(* IEC 61131-3 sources: ics/BLR1_PhoenixContact/BLR1_AXC1050_21/LogicalPOUs/AIO, 3 files *)

(* ---- SensorFB.ST ---- *)
(*@PROPERTIES_EX@
TYPE: POU
LOCALE: 0
IEC_LANGUAGE: ST
PLC_TYPE: independent
PROC_TYPE: independent
GROUP: AIO.FB
*)
(*@KEY@:DESCRIPTION*)

(*@KEY@:END_DESCRIPTION*)
FUNCTION_BLOCK SensorFB

(*Group:Default*)

VAR_IN_OUT
    Snsr_strct :	SNSR;
END_VAR

VAR
    RealValue :	REAL;
    bar_kgf :	REAL;
END_VAR

VAR_IN_OUT
    Buff :	SNSR_BUFF;
END_VAR

VAR
    SumValue :	REAL;
    y :	INT;
    INIT :	BOOL;
    FltrValue :	REAL;
    x :	INT;
END_VAR

VAR_OUTPUT
    Event :	SNSR_EVENT;
END_VAR

VAR_IN_OUT
    Aux_strct :	SNSR_MISC;
END_VAR

VAR_EXTERNAL
    TICK_100MS_PLS :	BOOL;
END_VAR

(*@KEY@: WORKSHEET
NAME: SensorFB
IEC_LANGUAGE: ST
*)

(*============================================================================*)
(*Fault operation & converting PIW to real value*)
(*============================================================================*)
IF (Snsr_strct.PIW < 0) OR (Snsr_strct.PIW > Snsr_strct.ADC_Range) OR
    Snsr_strct.CW.ExtFault OR (Snsr_strct.DiagCode > word#16#8000) THEN         (*Snsr_strct Failed*)
    Snsr_strct.SW.Fault:= TRUE;
    RealValue:= 0.0;
ELSE                                                                            (*Snsr_strct OK*)
    IF Snsr_strct.ADC_Range <= 0 THEN
        Snsr_strct.ADC_Range:= 1;
    END_IF;
    Snsr_strct.SW.Fault:= FALSE;
    RealValue:= (Snsr_strct.Ymax - Snsr_strct.Ymin) * bar_kgf *
        INT_TO_REAL(Snsr_strct.PIW) / INT_TO_REAL(Snsr_strct.ADC_Range) +
        Snsr_strct.Ymin ;
END_IF;

(*============================================================================*)
(*Converting from bar to kgf/sm2*)
(*============================================================================*)
IF Snsr_strct.CW.bar_kgf THEN
    bar_kgf:= 1.0197;
ELSE
    bar_kgf:= 1.0;
END_IF;

(*============================================================================*)
(*SMA filter operation*)
(*============================================================================*)
IF INIT THEN
    IF TICK_100MS_PLS THEN
        Aux_strct.SamplingTickCount:= Aux_strct.SamplingTickCount + 1;
    END_IF;
ELSE
    Aux_strct.SamplingTickCount:= 0;
END_IF;

IF Snsr_strct.CW.FltrEn THEN
    IF NOT INIT THEN                                                            (*Initialization*)
        FOR y:= 0 TO 9 DO
            Buff[y]:= RealValue;
            SumValue:= SumValue + Buff[y];
        END_FOR;
        INIT:= TRUE;
    ELSE
        IF Aux_strct.SamplingTickCount >= (Snsr_strct.SamplingTime * 10) THEN   (*Buffer shIFting AND changing last element*)
            FOR y:= 0 TO 8 DO
                x:= y + 1;
                Buff[y]:= Buff[x];
            END_FOR;
            Buff[9]:= RealValue;
            SumValue:= SumValue + RealValue - Buff[0];
            Aux_strct.SamplingTickCount:= 0;
        END_IF;
        FltrValue:= SumValue / 10.0;
    END_IF;
ELSE
    INIT:= FALSE;
    SumValue:= 0.0;
    FltrValue:= 0.0;
END_IF;

(*============================================================================*)
(*Snsr_strct output values states*)
(*============================================================================*)
IF Snsr_strct.CW.SimEn THEN                                                     (*Simulated output value*)
    Snsr_strct.RealValue:= Snsr_strct.SimValue;
ELSIF Snsr_strct.CW.FltrEn THEN                                                 (*Filtered output value*)
    Snsr_strct.RealValue:= FltrValue;
ELSE                                                                            (*Real output value*)
    Snsr_strct.RealValue:= RealValue;
END_IF;

Snsr_strct.IntValue:= REAL_TO_INT(Snsr_strct.RealValue * 100.0);

(*============================================================================*)
(*Limits operation*)
(*============================================================================*)
IF Snsr_strct.CW.LimEn THEN
    IF (Snsr_strct.RealValue > (Snsr_strct.HH + (Snsr_strct.DeadBand / 2.0))) and
        not Snsr_strct.SW.HH_alarm  THEN
        IF TICK_100MS_PLS THEN
            Aux_strct.HHTopDelayCount:= Aux_strct.HHTopDelayCount + 1;
        END_IF;
        IF Aux_strct.HHTopDelayCount > (Snsr_strct.LimDelay * 10) THEN
            Snsr_strct.SW.HH_alarm:= true;
        END_IF;
    ELSE
        Aux_strct.HHTopDelayCount:= 0;
    END_IF;

    IF (Snsr_strct.RealValue < (Snsr_strct.HH - (Snsr_strct.DeadBand / 2.0))) and
        Snsr_strct.SW.HH_alarm THEN
        IF TICK_100MS_PLS THEN
            Aux_strct.HHBotDelayCount:= Aux_strct.HHBotDelayCount + 1;
        END_IF;
        IF Aux_strct.HHBotDelayCount > (Snsr_strct.LimDelay * 10) THEN
            Snsr_strct.SW.HH_alarm:= false;
        END_IF;
    ELSE
        Aux_strct.HHBotDelayCount:= 0;
    END_IF;

    IF (Snsr_strct.RealValue > (Snsr_strct.HL + (Snsr_strct.DeadBand / 2.0))) and
        not Snsr_strct.SW.HL_alarm THEN
        IF TICK_100MS_PLS THEN
            Aux_strct.HLTopDelayCount:= Aux_strct.HLTopDelayCount + 1;
        END_IF;
        IF Aux_strct.HLTopDelayCount > (Snsr_strct.LimDelay * 10) THEN
            Snsr_strct.SW.HL_alarm:= true;
        END_IF;
    ELSE
        Aux_strct.HLTopDelayCount:= 0;
    END_IF;

    IF (Snsr_strct.RealValue < (Snsr_strct.HL - (Snsr_strct.DeadBand / 2.0))) and
        Snsr_strct.SW.HL_alarm THEN
        IF TICK_100MS_PLS THEN
            Aux_strct.HLBotDelayCount:= Aux_strct.HLBotDelayCount + 1;
        END_IF;
        IF Aux_strct.HLBotDelayCount > (Snsr_strct.LimDelay * 10) THEN
            Snsr_strct.SW.HL_alarm:= false;
        END_IF;
    ELSE
        Aux_strct.HLBotDelayCount:= 0;
    END_IF;

    IF (Snsr_strct.RealValue < (Snsr_strct.LH - (Snsr_strct.DeadBand / 2.0))) and
        not Snsr_strct.SW.LH_alarm THEN
        IF TICK_100MS_PLS THEN
            Aux_strct.LHTopDelayCount:= Aux_strct.LHTopDelayCount + 1;
        END_IF;
        IF Aux_strct.LHTopDelayCount > (Snsr_strct.LimDelay * 10) THEN
            Snsr_strct.SW.LH_alarm:= true;
        END_IF;
    ELSE
        Aux_strct.LHTopDelayCount:= 0;
    END_IF;

    IF (Snsr_strct.RealValue > (Snsr_strct.LH + (Snsr_strct.DeadBand / 2.0))) and
        Snsr_strct.SW.LH_alarm THEN
        IF TICK_100MS_PLS THEN
            Aux_strct.LHBotDelayCount:= Aux_strct.LHBotDelayCount + 1;
        END_IF;
        IF Aux_strct.LHBotDelayCount > (Snsr_strct.LimDelay * 10) THEN
            Snsr_strct.SW.LH_alarm:= false;
        END_IF;
    ELSE
        Aux_strct.LHBotDelayCount:= 0;
    END_IF;

    IF (Snsr_strct.RealValue < (Snsr_strct.LL - (Snsr_strct.DeadBand / 2.0))) and
        not Snsr_strct.SW.LL_alarm THEN
        IF TICK_100MS_PLS THEN
            Aux_strct.LLTopDelayCount:= Aux_strct.LLTopDelayCount + 1;
        END_IF;
        IF Aux_strct.LLTopDelayCount > (Snsr_strct.LimDelay * 10) THEN
            Snsr_strct.SW.LL_alarm:= true;
        END_IF;
    ELSE
        Aux_strct.LLTopDelayCount:= 0;
    END_IF;

    IF (Snsr_strct.RealValue > (Snsr_strct.LL + (Snsr_strct.DeadBand / 2.0))) and
        Snsr_strct.SW.LL_alarm THEN
        IF TICK_100MS_PLS THEN
            Aux_strct.LLBotDelayCount:= Aux_strct.LLBotDelayCount + 1;
        END_IF;
        IF Aux_strct.LLBotDelayCount > (Snsr_strct.LimDelay * 10) THEN
            Snsr_strct.SW.LL_alarm:= false;
        END_IF;
    ELSE
        Aux_strct.LLBotDelayCount:= 0;
    END_IF;

ELSE
    Aux_strct.HHTopDelayCount:= 0;
    Aux_strct.HHBotDelayCount:= 0;

    Aux_strct.HLTopDelayCount:= 0;
    Aux_strct.HLBotDelayCount:= 0;

    Aux_strct.LHTopDelayCount:= 0;
    Aux_strct.LHBotDelayCount:= 0;

    Aux_strct.LLTopDelayCount:= 0;
    Aux_strct.LLBotDelayCount:= 0;

    Snsr_strct.SW.HH_alarm:= FALSE;
    Snsr_strct.SW.HL_alarm:= FALSE;
    Snsr_strct.SW.LH_alarm:= FALSE;
    Snsr_strct.SW.LL_alarm:= FALSE;
END_IF;

(*============================================================================*)
(*Sensor Pulse Events*)
(*============================================================================*)

Event.Fault:= false;
IF Snsr_strct.SW.Fault and not Aux_strct.EVENT_1 THEN
    Event.Fault:= true;
    Aux_strct.EVENT_1:= true;
ELSIF not Snsr_strct.SW.Fault THEN
    Aux_strct.EVENT_1:= false;
END_IF;

Event.HH:= false;
IF Snsr_strct.SW.HH_alarm and not Aux_strct.EVENT_2 THEN
    Event.HH:= true;
    Aux_strct.EVENT_2:= true;
ELSIF not Snsr_strct.SW.HH_alarm THEN
    Aux_strct.EVENT_2:= false;
END_IF;

Event.HL:= false;
IF Snsr_strct.SW.HL_alarm and not Aux_strct.EVENT_3 THEN
    Event.HL:= true;
    Aux_strct.EVENT_3:= true;
ELSIF not Snsr_strct.SW.HL_alarm THEN
    Aux_strct.EVENT_3:= false;
END_IF;

Event.LH:= false;
IF Snsr_strct.SW.LH_alarm and not Aux_strct.EVENT_4 THEN
    Event.LH:= true;
    Aux_strct.EVENT_4:= true;
ELSIF not Snsr_strct.SW.LH_alarm THEN
    Aux_strct.EVENT_4:= false;
END_IF;

Event.LL:= false;
IF Snsr_strct.SW.LL_alarm and not Aux_strct.EVENT_5 THEN
    Event.LL:= true;
    Aux_strct.EVENT_5:= true;
ELSIF not Snsr_strct.SW.LL_alarm THEN
    Aux_strct.EVENT_5:= false;
END_IF;

(*@KEY@: END_WORKSHEET *)
END_FUNCTION_BLOCK

(* ---- AI.ST ---- *)
(*@PROPERTIES_EX@
TYPE: POU
LOCALE: 0
IEC_LANGUAGE: ST
PLC_TYPE: independent
PROC_TYPE: independent
GROUP: AIO
*)
(*@KEY@:DESCRIPTION*)

(*@KEY@:END_DESCRIPTION*)
PROGRAM AI

(*Group:NewGroup*)

VAR_EXTERNAL
	AI :	SENSOR;
	A04_IN0 :	INT;
	A04_IN1 :	INT;
	A04_IN2 :	INT;
	A04_IN3 :	INT;
	A04_IN4 :	INT;
	A04_IN5 :	INT;
	A04_IN6 :	INT;
	A04_IN7 :	INT;
	A05_IN0 :	INT;
	A05_IN1 :	INT;
	A05_IN2 :	INT;
	A05_IN3 :	INT;
	A05_IN4 :	INT;
	A05_IN5 :	INT;
	A05_IN6 :	INT;
	A05_IN7 :	INT;
	A06_IN0 :	INT;
	A06_IN1 :	INT;
	A06_IN2 :	INT;
	A06_IN3 :	INT;
	A06_IN4 :	INT;
	A06_IN5 :	INT;
END_VAR

VAR
	SensorsFB :	SensorFB;
	i :	INT;
	AI_Buff :	SENSOR_BUFF;
END_VAR

VAR_EXTERNAL
	AI_Event :	SENSOR_EVENT;
	A16_IN0 :	INT;
	A16_IN1 :	INT;
	A16_IN2 :	INT;
	A16_IN3 :	INT;
	A16_IN4 :	INT;
	A16_IN5 :	INT;
	A16_IN6 :	INT;
	A16_IN7 :	INT;
	A17_IN0 :	INT;
	A17_IN1 :	INT;
	A17_IN2 :	INT;
	A17_IN3 :	INT;
	A17_IN4 :	INT;
	A17_IN5 :	INT;
	A17_IN6 :	INT;
	A17_IN7 :	INT;
	A18_IN0 :	INT;
	A18_IN1 :	INT;
	A18_IN2 :	INT;
	A18_IN3 :	INT;
	A18_IN4 :	INT;
	A18_IN5 :	INT;
	A18_IN6 :	INT;
	A18_IN7 :	INT;
	A19_IN0 :	INT;
	A19_IN1 :	INT;
	A19_IN2 :	INT;
	A19_IN3 :	INT;
	A19_IN4 :	INT;
	A19_IN5 :	INT;
	A19_IN6 :	INT;
	A19_IN7 :	INT;
	A110_IN0 :	INT;
	A110_IN1 :	INT;
	A110_IN2 :	INT;
	A110_IN3 :	INT;
	A110_IN4 :	INT;
	A110_IN5 :	INT;
	A110_IN6 :	INT;
	A110_IN7 :	INT;
	A111_IN0 :	INT;
	A111_IN1 :	INT;
	A111_IN2 :	INT;
	A111_IN3 :	INT;
	A111_IN4 :	INT;
	A111_IN5 :	INT;
	A111_IN6 :	INT;
	A111_IN7 :	INT;
	A112_IN0 :	INT;
	A112_IN1 :	INT;
	A112_IN2 :	INT;
	A112_IN3 :	INT;
	A112_IN4 :	INT;
	A112_IN5 :	INT;
	A112_IN6 :	INT;
	A112_IN7 :	INT;
	A113_IN0 :	INT;
	A113_IN1 :	INT;
	A113_IN2 :	INT;
	A113_IN3 :	INT;
	A113_IN4 :	INT;
	A113_IN5 :	INT;
	A113_IN6 :	INT;
	A113_IN7 :	INT;
	A114_IN0 :	INT;
	A114_IN1 :	INT;
	A114_IN2 :	INT;
	A114_IN3 :	INT;
	A114_IN4 :	INT;
	A114_IN5 :	INT;
	A114_IN6 :	INT;
	A114_IN7 :	INT;
	A115_IN0 :	INT;
	A115_IN1 :	INT;
	A115_IN2 :	INT;
	A115_IN3 :	INT;
	A115_IN4 :	INT;
	A115_IN5 :	INT;
	A115_IN6 :	INT;
	A115_IN7 :	INT;
	A06_IN7 :	INT;
	A06_IN6 :	INT;
	AI_AUX :	SENSOR_MISC;
	SlvData_RSUNI_2 :	MBRTU_SlvData;
END_VAR

VAR
	MB_TO_REAL :	MB_TO_REAL;
END_VAR

(*@KEY@: WORKSHEET
NAME: AI
IEC_LANGUAGE: ST
*)
(*============================================================================*)
	(*PT5100 Pump 5.1 input pressure sensor*)
(*============================================================================*)
AI[0].PIW:= A04_IN0;
AI[0].DiagCode:= int_to_word(A04_IN0);
AI[0].CW.bar_kgf:= true;

(*============================================================================*)
	(*PT5101 Pump 5.1 output pressure sensor*)
(*============================================================================*)
AI[1].PIW:= A04_IN1;
AI[1].DiagCode:= int_to_word(A04_IN1);
AI[1].CW.bar_kgf:= true;

(*============================================================================*)
	(*PT5200 Pump 5.2 input pressure sensor*)
(*============================================================================*)
AI[2].PIW:= A04_IN2;
AI[2].DiagCode:= int_to_word(A04_IN2);
AI[2].CW.bar_kgf:= true;

(*============================================================================*)
	(*PT5201 Pump 5.2 output pressure sensor*)
(*============================================================================*)
AI[3].PIW:= A04_IN3;
AI[3].DiagCode:= int_to_word(A04_IN3);
AI[3].CW.bar_kgf:= true;

(*============================================================================*)
	(*PT5300 Pump 5.3 input pressure sensor*)
(*============================================================================*)
AI[4].PIW:= A04_IN4;
AI[4].DiagCode:= int_to_word(A04_IN4);
AI[4].CW.bar_kgf:= true;

(*============================================================================*)
	(*PT5301 Pump 5.3 output pressure sensor*)
(*============================================================================*)
AI[5].PIW:= A04_IN5;
AI[5].DiagCode:= int_to_word(A04_IN5);
AI[5].CW.bar_kgf:= true;

(*============================================================================*)
	(*PT009  Pumps 5 input collector pressure sensor*)
(*============================================================================*)
AI[6].PIW:= A04_IN6;
AI[6].DiagCode:= int_to_word(A04_IN6);
AI[6].CW.bar_kgf:= true;

(*============================================================================*)
	(*PT010  Pumps 5 output collector pressure sensor*)
(*============================================================================*)
AI[7].PIW:= A04_IN7;
AI[7].DiagCode:= int_to_word(A04_IN7);
AI[7].CW.bar_kgf:= true;

(*============================================================================*)
	(*TT001  Boiler 1.1 output temperature sensor*)
(*============================================================================*)
AI[8].PIW:= A05_IN0;
AI[8].DiagCode:= int_to_word(A05_IN0);
AI[8].CW.bar_kgf:= false;

(*============================================================================*)
	(*PT002  Boiler 1.1 output pressure sensor*)
(*============================================================================*)
AI[9].PIW:= A05_IN1;
AI[9].DiagCode:= int_to_word(A05_IN1);
AI[9].CW.bar_kgf:= true;

(*============================================================================*)
	(*TT003  Boiler 1.1 input temperature sensor*)
(*============================================================================*)
AI[10].PIW:= A05_IN2;
AI[10].DiagCode:= int_to_word(A05_IN2);
AI[10].ADC_Range:= 30000;
AI[10].CW.bar_kgf:= false;

(*============================================================================*)
	(*PT004  Boiler 1.1 input pressure sensor*)
(*============================================================================*)
AI[11].PIW:= A05_IN3;
AI[11].DiagCode:= int_to_word(A05_IN3);
AI[11].CW.bar_kgf:= true;

(*============================================================================*)
	(*TT005  Boiler 1.2 output temperature sensor*)
(*============================================================================*)
AI[12].PIW:= A05_IN4;
AI[12].DiagCode:= int_to_word(A05_IN4);
AI[12].CW.bar_kgf:= false;

(*============================================================================*)
	(*PT006  Boiler 1.2 output pressure sensor*)
(*============================================================================*)
AI[13].PIW:= A05_IN5;
AI[13].DiagCode:= int_to_word(A05_IN5);
AI[13].CW.bar_kgf:= true;

(*============================================================================*)
	(*TT007  Boiler 1.2 input temperature sensor*)
(*============================================================================*)
AI[14].PIW:= A05_IN6;
AI[14].DiagCode:= int_to_word(A05_IN6);
AI[14].CW.bar_kgf:= false;

(*============================================================================*)
	(*PT008  Boiler 1.2 input pressure sensor*)
(*============================================================================*)
AI[15].PIW:= A05_IN7;
AI[15].DiagCode:= int_to_word(A05_IN7);
AI[15].CW.bar_kgf:= true;

(*============================================================================*)
	(*UZ5100AO FC actual frequency*)
(*============================================================================*)
AI[16].PIW:= A06_IN0;
AI[16].DiagCode:= int_to_word(A06_IN0);
AI[16].CW.bar_kgf:= false;
AI[16].Ymin:= 0.0;
AI[16].Ymax:= 50.0;

(*============================================================================*)
	(*UZ5200AO FC actual frequency*)
(*============================================================================*)
AI[17].PIW:= A06_IN1;
AI[17].DiagCode:= int_to_word(A06_IN1);
AI[17].CW.bar_kgf:= false;
AI[17].Ymin:= 0.0;
AI[17].Ymax:= 50.0;

(*============================================================================*)
	(*UZ5300AO FC actual frequency*)
(*============================================================================*)
AI[18].PIW:= A06_IN2;
AI[18].DiagCode:= int_to_word(A06_IN2);
AI[18].CW.bar_kgf:= false;
AI[18].Ymin:= 0.0;
AI[18].Ymax:= 50.0;

(*============================================================================*)
	(*PT011  Boiler 1.1 gas pressure sensor*)
(*============================================================================*)
AI[19].PIW:= A06_IN3;
AI[19].DiagCode:= int_to_word(A06_IN3);
AI[19].CW.bar_kgf:= true;

(*============================================================================*)
	(*PT012  Boiler 1.2 gas pressure sensor*)
(*============================================================================*)
AI[20].PIW:= A06_IN4;
AI[20].DiagCode:= int_to_word(A06_IN4);
AI[20].CW.bar_kgf:= true;

(*============================================================================*)
	(*TT013 Heat carrier feed temperature sensor*)
(*============================================================================*)
AI[21].PIW:= A06_IN5;
AI[21].DiagCode:= int_to_word(A06_IN5);
AI[21].CW.bar_kgf:= false;

(*============================================================================*)
	(*Reserve*)
(*============================================================================*)
AI[22].PIW:= A06_IN6;
AI[22].DiagCode:= int_to_word(A06_IN6);
AI[22].CW.bar_kgf:= false;

(*============================================================================*)
	(*Reserve*)
(*============================================================================*)
AI[23].PIW:= A06_IN7;
AI[23].DiagCode:= int_to_word(A06_IN7);
AI[23].CW.bar_kgf:= false;

(*============================================================================*)
	(*TT1106 Boiler 1.1 smoke temperature sensor*)
(*============================================================================*)
AI[24].PIW:= A16_IN0;
AI[24].DiagCode:= int_to_word(A16_IN0);
AI[24].CW.bar_kgf:= false;

(*============================================================================*)
	(*TT1206 Boiler 1.2 smoke temperature sensor*)
(*============================================================================*)
AI[25].PIW:= A16_IN1;
AI[25].DiagCode:= int_to_word(A16_IN1);
AI[25].CW.bar_kgf:= false;

(*============================================================================*)
	(*TT1306 Boiler 1.3 smoke temperature sensor*)
(*============================================================================*)
AI[26].PIW:= A16_IN2;
AI[26].DiagCode:= int_to_word(A16_IN2);
AI[26].CW.bar_kgf:= false;

(*============================================================================*)
	(*PT3-2 Gas pressure sensor (for boiler 1.3)*)
(*============================================================================*)
AI[27].PIW:= A16_IN3;
AI[27].DiagCode:= int_to_word(A16_IN3);
AI[27].CW.bar_kgf:= true;

(*============================================================================*)
	(*TT009 Boiler 1.3 output water temperature sensor*)
(*============================================================================*)
AI[28].PIW:= A16_IN4;
AI[28].DiagCode:= int_to_word(A16_IN4);
AI[28].CW.bar_kgf:= false;

(*============================================================================*)
	(*PT015 Boiler 1.3 output water pressure sensor*)
(*============================================================================*)
AI[29].PIW:= A16_IN5;
AI[29].DiagCode:= int_to_word(A16_IN5);
AI[29].CW.bar_kgf:= true;

(*============================================================================*)
	(*TT011 Boiler 1.3 input temperature sensor*)
(*============================================================================*)
AI[30].PIW:= A16_IN6;
AI[30].DiagCode:= int_to_word(A16_IN6);
AI[30].CW.bar_kgf:= false;

(*============================================================================*)
	(*PT012 Boiler 1.3 input pressure sensor*)
(*============================================================================*)
AI[31].PIW:= A16_IN7;
AI[31].DiagCode:= int_to_word(A16_IN7);
AI[31].CW.bar_kgf:= true;

(*============================================================================*)
	(*PT014 Boilers 1.x output water pressure sensor*)
(*============================================================================*)
AI[32].PIW:= A17_IN0;
AI[32].DiagCode:= int_to_word(A17_IN0);
AI[32].CW.bar_kgf:= true;

(*============================================================================*)
	(*TT2103 Boiler 2.1 smoke temperature sensor*)
(*============================================================================*)
AI[33].PIW:= A17_IN1;
AI[33].DiagCode:= int_to_word(A17_IN1);
AI[33].CW.bar_kgf:= false;

(*============================================================================*)
	(*PT2105 Boiler 2.1 output pressure sensor*)
(*============================================================================*)
AI[34].PIW:= A17_IN2;
AI[34].DiagCode:= int_to_word(A17_IN2);
AI[34].CW.bar_kgf:= true;

(*============================================================================*)
	(*TT2107 Boiler 2.1 output temperature sensor*)
(*============================================================================*)
AI[35].PIW:= A17_IN3;
AI[35].DiagCode:= int_to_word(A17_IN3);
AI[35].CW.bar_kgf:= false;

(*============================================================================*)
	(*PT4-2 Gas pressure sensor (for boiler 2.1)*)
(*============================================================================*)
AI[36].PIW:= A17_IN4;
AI[36].DiagCode:= int_to_word(A17_IN4);
AI[36].CW.bar_kgf:= true;

(*============================================================================*)
	(*TT2203 Boiler 2.2 smoke temperature sensor*)
(*============================================================================*)
AI[37].PIW:= A17_IN5;
AI[37].DiagCode:= int_to_word(A17_IN5);
AI[37].CW.bar_kgf:= false;

(*============================================================================*)
	(*PT2205 Boiler 2.2 output pressure sensor*)
(*============================================================================*)
AI[38].PIW:= A17_IN6;
AI[38].DiagCode:= int_to_word(A17_IN6);
AI[38].CW.bar_kgf:= true;

(*============================================================================*)
	(*TT2207 Boiler 2.2 output temperature sensor*)
(*============================================================================*)
AI[39].PIW:= A17_IN7;
AI[39].DiagCode:= int_to_word(A17_IN7);
AI[39].CW.bar_kgf:= false;

(*============================================================================*)
	(*PT5-2 Gas pressure sensor (for boiler 2.2)*)
(*============================================================================*)
AI[40].PIW:= A18_IN0;
AI[40].DiagCode:= int_to_word( A18_IN0);
AI[40].CW.bar_kgf:= true;

(*============================================================================*)
	(*TT2001 Boilers 2.x input temperature sensor*)
(*============================================================================*)
AI[41].PIW:= A18_IN1;
AI[41].DiagCode:= int_to_word(A18_IN1);
AI[41].CW.bar_kgf:= false;

(*============================================================================*)
	(*PT2002 Boilers 2.x input pressure sensor*)
(*============================================================================*)
AI[42].PIW:= A18_IN2;
AI[42].DiagCode:= int_to_word(A18_IN2);
AI[42].CW.bar_kgf:= true;

(*============================================================================*)
	(*TT2003 Boilers 2.x output temperature sensor*)
(*============================================================================*)
AI[43].PIW:= A18_IN3;
AI[43].DiagCode:= int_to_word(A18_IN3);
AI[43].CW.bar_kgf:= false;

(*============================================================================*)
	(*PT2004 Boilers 2.x output pressure sensor*)
(*============================================================================*)
AI[44].PIW:= A18_IN4;
AI[44].DiagCode:= int_to_word(A18_IN4);
AI[44].CW.bar_kgf:= true;

(*============================================================================*)
	(*PT3000 Pumps 3.x input collector pressure sensor*)
(*============================================================================*)
AI[45].PIW:= A18_IN5;
AI[45].DiagCode:= int_to_word(A18_IN5);
AI[45].CW.bar_kgf:= true;

(*============================================================================*)
	(*PT3100 Pump 3.1 input pressure sensor*)
(*============================================================================*)
AI[46].PIW:= A18_IN6;
AI[46].DiagCode:= int_to_word(A18_IN6);
AI[46].CW.bar_kgf:= true;

(*============================================================================*)
	(*PT3101 Pump 3.1 output pressure sensor*)
(*============================================================================*)
AI[47].PIW:= A18_IN7;
AI[47].DiagCode:= int_to_word(A18_IN7);
AI[47].CW.bar_kgf:= true;

(*============================================================================*)
	(*UZ3100AO FC actual frequency*)
(*============================================================================*)
AI[48].PIW:= A19_IN0;
AI[48].DiagCode:= int_to_word(A19_IN0);
AI[48].CW.bar_kgf:= false;
AI[48].Ymin:= 0.0;
AI[48].Ymax:= 50.0;

(*============================================================================*)
	(*PT3200 Pump 3.2 input pressure sensor*)
(*============================================================================*)
AI[49].PIW:= A19_IN1;
AI[49].DiagCode:= int_to_word(A19_IN1);
AI[49].CW.bar_kgf:= true;

(*============================================================================*)
	(*PT3201 Pump 3.2 output pressure sensor*)
(*============================================================================*)
AI[50].PIW:= A19_IN2;
AI[50].DiagCode:= int_to_word(A19_IN2);
AI[50].CW.bar_kgf:= true;

(*============================================================================*)
	(*UZ3200AO FC actual frequency*)
(*============================================================================*)
AI[51].PIW:= A19_IN3;
AI[51].DiagCode:= int_to_word(A19_IN3);
AI[51].CW.bar_kgf:= false;
AI[51].Ymin:= 0.0;
AI[51].Ymax:= 50.0;

(*============================================================================*)
	(*PT3300 Pump 3.3 input pressure sensor*)
(*============================================================================*)
AI[52].PIW:= A19_IN4;
AI[52].DiagCode:= int_to_word(A19_IN4);
AI[52].CW.bar_kgf:= true;

(*============================================================================*)
	(*PT3301 Pump 3.3 output pressure sensor*)
(*============================================================================*)
AI[53].PIW:= A19_IN5;
AI[53].DiagCode:= int_to_word(A19_IN5);
AI[53].CW.bar_kgf:= true;

(*============================================================================*)
	(*UZ3300AO FC actual frequency*)
(*============================================================================*)
AI[54].PIW:= A19_IN6;
AI[54].DiagCode:= int_to_word(A19_IN6);
AI[54].CW.bar_kgf:= false;
AI[54].Ymin:= 0.0;
AI[54].Ymax:= 50.0;

(*============================================================================*)
	(*PT3004 Pumps 3.x output collector pressure sensor*)
(*============================================================================*)
AI[55].PIW:= A19_IN7;
AI[55].DiagCode:= int_to_word(A19_IN7);
AI[55].CW.bar_kgf:= true;

(*============================================================================*)
	(*TT3005 Pumps 3.x output collector temperature sensor*)
(*============================================================================*)
AI[56].PIW:= A110_IN0;
AI[56].DiagCode:= int_to_word(A110_IN0);
AI[56].CW.bar_kgf:= false;

(*============================================================================*)
	(*TT5001 Filter A4 input temperature sensor*)
(*============================================================================*)
AI[57].PIW:= A110_IN1;
AI[57].DiagCode:= int_to_word(A110_IN1);
AI[57].CW.bar_kgf:= false;

(*============================================================================*)
	(*PT5002 Filter A4 input pressure sensor*)
(*============================================================================*)
AI[58].PIW:= A110_IN2;
AI[58].DiagCode:= int_to_word(A110_IN2);
AI[58].CW.bar_kgf:= true;

(*============================================================================*)
	(*PT5005 Filter A4 output pressure sensor*)
(*============================================================================*)
AI[59].PIW:= A110_IN3;
AI[59].DiagCode:= int_to_word(A110_IN3);
AI[59].CW.bar_kgf:= true;

(*============================================================================*)
	(*TT7001*)
(*============================================================================*)
AI[60].PIW:= A110_IN4;
AI[60].DiagCode:= int_to_word(A110_IN4);
AI[60].CW.bar_kgf:= false;

(*============================================================================*)
	(*PT7003 Feed T12 pressure sensor (before accounting unit)*)
(*============================================================================*)
AI[61].PIW:= A110_IN5;
AI[61].DiagCode:= int_to_word(A110_IN5);
AI[61].CW.bar_kgf:= true;

(*============================================================================*)
	(*TT7005 External temperature sensor*)
(*============================================================================*)
AI[62].PIW:= A110_IN6;
AI[62].DiagCode:= int_to_word(A110_IN6);
AI[62].CW.bar_kgf:= false;

(*============================================================================*)
	(*TT7006 Internal temperature sensor*)
(*============================================================================*)
AI[63].PIW:= A110_IN7;
AI[63].DiagCode:= int_to_word(A110_IN7);
AI[63].CW.bar_kgf:= false;

(*============================================================================*)
	(*TT8019 Hot water feed temperature sensor*)
(*============================================================================*)
AI[64].PIW:= A111_IN0;
AI[64].DiagCode:= int_to_word(A111_IN0);
AI[64].CW.bar_kgf:= false;

(*============================================================================*)
	(*PT8017 Hot water feed pressure sensor*)
(*============================================================================*)
AI[65].PIW:= A111_IN1;
AI[65].DiagCode:= int_to_word(A111_IN0);
AI[65].CW.bar_kgf:= true;

(*============================================================================*)
	(*PT8007 Heat exchanger 8 cold water input pressure sensor*)
(*============================================================================*)
AI[66].PIW:= A111_IN2;
AI[66].DiagCode:= int_to_word(A111_IN2);
AI[66].CW.bar_kgf:= true;

(*============================================================================*)
	(*TT8008 Heat exchanger 8 cold water input temperature sensor*)
(*============================================================================*)
AI[67].PIW:= A111_IN3;
AI[67].DiagCode:= int_to_word(A111_IN3);
AI[67].CW.bar_kgf:= false;

(*============================================================================*)
	(*TT8001 Pipeline T4 hot water input temperature sensor*)
(*============================================================================*)
AI[68].PIW:= A111_IN4;
AI[68].DiagCode:= int_to_word(A111_IN4);
AI[68].CW.bar_kgf:= false;

(*============================================================================*)
	(*PT8002 Pipeline T4 hot water input pressure sensor*)
(*============================================================================*)
AI[69].PIW:= A111_IN5;
AI[69].DiagCode:= int_to_word(A111_IN5);
AI[69].CW.bar_kgf:= true;

(*============================================================================*)
	(*PT8020 Pumps 6.x input pressure sensor*)
(*============================================================================*)
AI[70].PIW:= A111_IN6;
AI[70].DiagCode:= int_to_word(A111_IN6);
AI[70].CW.bar_kgf:= true;

(*============================================================================*)
	(*PT8021 Pumps 6.x output pressure sensor*)
(*============================================================================*)
AI[71].PIW:= A111_IN7;
AI[71].DiagCode:= int_to_word(A111_IN7);
AI[71].CW.bar_kgf:= true;

(*============================================================================*)
	(*UZ6100AO FC actual frequency*)
(*============================================================================*)
AI[72].PIW:= A112_IN0;
AI[72].DiagCode:= int_to_word(A112_IN0);
AI[72].CW.bar_kgf:= false;
AI[72].Ymin:= 0.0;
AI[72].Ymax:= 50.0;

(*============================================================================*)
	(*UZ6200AO FC actual frequency*)
(*============================================================================*)
AI[73].PIW:= A112_IN1;
AI[73].DiagCode:= int_to_word(A112_IN1);
AI[73].CW.bar_kgf:= false;
AI[73].Ymin:= 0.0;
AI[73].Ymax:= 50.0;

(*============================================================================*)
	(*TT9008 Heat exchanger 9 hot water output temperature sensor*)
(*============================================================================*)
AI[74].PIW:= A112_IN2;
AI[74].DiagCode:= int_to_word(A112_IN2);
AI[74].CW.bar_kgf:= false;

(*============================================================================*)
	(*PT9010 Heat exchanger 5 supply water input pressure sensor*)
(*============================================================================*)
AI[75].PIW:= A112_IN3;
AI[75].DiagCode:= int_to_word(A112_IN3);
AI[75].CW.bar_kgf:= true;

(*============================================================================*)
	(*PT0019 Water preparation unit output pressure sensor*)
(*============================================================================*)
AI[76].PIW:= A112_IN4;
AI[76].DiagCode:= int_to_word(A112_IN4);
AI[76].CW.bar_kgf:= true;

(*============================================================================*)
	(*PT0022 Cold water feed pressure sensor*)
(*============================================================================*)
AI[77].PIW:= A112_IN5;
AI[77].DiagCode:= int_to_word(A112_IN5);
AI[77].CW.bar_kgf:= true;

(*============================================================================*)
	(*TT0023 Cold water feed temperature sensor*)
(*============================================================================*)
AI[78].PIW:= A112_IN6;
AI[78].DiagCode:= int_to_word(A112_IN6);
AI[78].CW.bar_kgf:= false;

(*============================================================================*)
	(*PT0027 Return water pressure sensor*)
(*============================================================================*)
AI[79].PIW:= A112_IN7;
AI[79].DiagCode:= int_to_word(A112_IN7);
AI[79].CW.bar_kgf:= true;

(*============================================================================*)
	(*TT0028 Return water temperature sensor*)
(*============================================================================*)
AI[80].PIW:= A113_IN0;
AI[80].DiagCode:= int_to_word(A113_IN0);
AI[80].CW.bar_kgf:= false;

(*============================================================================*)
	(*PT0031 Feed water pressure sensor*)
(*============================================================================*)
AI[81].PIW:= A113_IN1;
AI[81].DiagCode:= int_to_word(A113_IN1);
AI[81].CW.bar_kgf:= true;

(*============================================================================*)
	(*TT0032 Feed water temperature sensor*)
(*============================================================================*)
AI[82].PIW:= A113_IN2;
AI[82].DiagCode:= int_to_word(A113_IN2);
AI[82].CW.bar_kgf:= false;

(*============================================================================*)
	(*PT0035 Return water pressure sensor*)
(*============================================================================*)
AI[83].PIW:= A113_IN3;
AI[83].DiagCode:= int_to_word(A113_IN3);
AI[83].CW.bar_kgf:= true;

(*============================================================================*)
	(*TT0036 Return water temperature sensor*)
(*============================================================================*)
AI[84].PIW:= A113_IN4;
AI[84].DiagCode:= int_to_word(A113_IN4);
AI[84].CW.bar_kgf:= false;

(*============================================================================*)
	(*PT0039 Feed water pressure sensor*)
(*============================================================================*)
AI[85].PIW:= A113_IN5;
AI[85].DiagCode:= int_to_word(A113_IN5);
AI[85].CW.bar_kgf:= true;

(*============================================================================*)
	(*TT0040 Feed water temperature sensor*)
(*============================================================================*)
AI[86].PIW:= A113_IN6;
AI[86].DiagCode:= int_to_word(A113_IN6);
AI[86].CW.bar_kgf:= false;

(*============================================================================*)
	(*PT0041 Hot water return pressure sensor*)
(*============================================================================*)
AI[87].PIW:= A113_IN7;
AI[87].DiagCode:= int_to_word(A113_IN7);
AI[87].CW.bar_kgf:= true;

(*============================================================================*)
	(*TT0042 Hot water return temperature sensor*)
(*============================================================================*)
AI[88].PIW:= A114_IN0;
AI[88].DiagCode:= int_to_word(A114_IN0);
AI[88].CW.bar_kgf:= false;

(*============================================================================*)
	(*PT0046 Hot water feed pressure sensor*)
(*============================================================================*)
AI[89].PIW:= A114_IN1;
AI[89].DiagCode:= int_to_word(A114_IN1);
AI[89].CW.bar_kgf:= true;

(*============================================================================*)
	(*TT0047 Hot water feed temperature sensor*)
(*============================================================================*)
AI[90].PIW:= A114_IN2;
AI[90].DiagCode:= int_to_word(A114_IN2);
AI[90].CW.bar_kgf:= false;

(*============================================================================*)
	(*TV7001 Valve actual position*)
(*============================================================================*)
AI[91].Ymin:= 0.0;
AI[91].Ymax:= 100.0;
AI[91].PIW:= A114_IN3;
AI[91].DiagCode:= int_to_word(A114_IN3);
AI[91].CW.bar_kgf:= false;

(*============================================================================*)
	(*TV8019 Valve actual position*)
(*============================================================================*)
AI[92].Ymin:= 0.0;
AI[92].Ymax:= 100.0;
AI[92].PIW:= A114_IN4;
AI[92].DiagCode:= int_to_word(A114_IN4);
AI[92].CW.bar_kgf:= false;

(*============================================================================*)
	(*TV9008 Valve actual position*)
(*============================================================================*)
AI[93].Ymin:= 0.0;
AI[93].Ymax:= 100.0;
AI[93].PIW:= A114_IN5;
AI[93].DiagCode:= int_to_word(A114_IN5);
AI[93].CW.bar_kgf:= false;

(*============================================================================*)
	(*FE Supply water flow*)
(*============================================================================*)
AI[94].PIW:= A114_IN6;
AI[94].DiagCode:= int_to_word(A114_IN6);
AI[94].CW.bar_kgf:= false;

(*============================================================================*)
	(*Reserve*)
(*============================================================================*)
AI[95].PIW:= A114_IN7;
AI[95].DiagCode:= int_to_word(A114_IN7);
AI[95].CW.bar_kgf:= false;

(*============================================================================*)
	(*Reserve*)
(*============================================================================*)
AI[96].PIW:= A115_IN0;
AI[96].DiagCode:= int_to_word(A115_IN0);
AI[96].CW.bar_kgf:= false;

(*============================================================================*)
	(*Reserve*)
(*============================================================================*)
AI[97].PIW:= A115_IN1;
AI[97].DiagCode:= int_to_word(A115_IN1);
AI[97].CW.bar_kgf:= false;

(*============================================================================*)
	(*Reserve*)
(*============================================================================*)
AI[98].PIW:= A115_IN2;
AI[98].DiagCode:= int_to_word(A115_IN2);
AI[98].CW.bar_kgf:= false;

(*============================================================================*)
	(*Reserve*)
(*============================================================================*)
AI[99].PIW:= A115_IN3;
AI[99].DiagCode:= int_to_word(A115_IN3);
AI[99].CW.bar_kgf:= false;

(*============================================================================*)
	(*Reserve*)
(*============================================================================*)
AI[100].PIW:= A115_IN4;
AI[100].DiagCode:= int_to_word(A115_IN4);
AI[100].CW.bar_kgf:= false;

(*============================================================================*)
	(*Reserve*)
(*============================================================================*)
AI[101].PIW:= A115_IN5;
AI[101].DiagCode:= int_to_word(A115_IN5);
AI[101].CW.bar_kgf:= false;

(*============================================================================*)
	(*Reserve*)
(*============================================================================*)
AI[102].PIW:= A115_IN6;
AI[102].DiagCode:= int_to_word(A115_IN6);
AI[102].CW.bar_kgf:= false;

(*============================================================================*)
	(*Reserve*)
(*============================================================================*)
AI[103].PIW:= A115_IN7;
AI[103].DiagCode:= int_to_word(A115_IN7);
AI[103].CW.bar_kgf:= false;

(*============================================================================*)
	(*Analog sensors FB processing*)
(*============================================================================*)
for i:= 0 to 103 do
	AI[i].ADC_Range:= 30000;
	SensorsFB(Snsr_strct:=AI[i],Buff:=AI_Buff[i],Aux_strct:=AI_AUX[i]);
	AI[i]:=SensorsFB.Snsr_strct;
	AI_Buff[i]:=SensorsFB.Buff;
	AI_Event[i]:=SensorsFB.Event;
	AI_AUX[i]:=SensorsFB.Aux_strct;
end_for;

(*============================================================================*)
	(*Boilers flowmeters (Promag)*)
(*============================================================================*)
MB_TO_REAL(LoWord:=SlvData_RSUNI_2[5][0],HiWord:=SlvData_RSUNI_2[5][1]);
AI[110].Ymax:=MB_TO_REAL.OUT;

MB_TO_REAL(LoWord:=SlvData_RSUNI_2[6][0],HiWord:=SlvData_RSUNI_2[6][1]);
AI[111].Ymax:=MB_TO_REAL.OUT;

MB_TO_REAL(LoWord:=SlvData_RSUNI_2[7][0],HiWord:=SlvData_RSUNI_2[7][1]);
AI[112].Ymax:=MB_TO_REAL.OUT;

MB_TO_REAL(LoWord:=SlvData_RSUNI_2[8][0],HiWord:=SlvData_RSUNI_2[8][1]);
AI[113].Ymax:=MB_TO_REAL.OUT;

MB_TO_REAL(LoWord:=SlvData_RSUNI_2[9][0],HiWord:=SlvData_RSUNI_2[9][1]);
AI[114].Ymax:=MB_TO_REAL.OUT;

(*============================================================================*)
	(*Supply flowmeter (US800)*)
(*============================================================================*)
MB_TO_REAL(LoWord:=SlvData_RSUNI_2[10][0],HiWord:=SlvData_RSUNI_2[10][1]);
AI[115].Ymax:=MB_TO_REAL.OUT;

(*============================================================================*)
	(*Flowmeters FB processing*)
(*============================================================================*)
for i:= 110 to 118 do
	AI[i].ADC_Range:= 1;
	AI[i].Ymin:= 0.0;
	AI[i].PIW:= 1;
	AI[i].CW.bar_kgf:= false;

	SensorsFB(Snsr_strct:=AI[i],Buff:=AI_Buff[i],Aux_strct:=AI_AUX[i]);
	AI[i]:=SensorsFB.Snsr_strct;
	AI_Buff[i]:=SensorsFB.Buff;
	AI_Event[i]:=SensorsFB.Event;
	AI_AUX[i]:=SensorsFB.Aux_strct;
end_for;
(*@KEY@: END_WORKSHEET *)
END_PROGRAM

(* ---- AO.ST ---- *)
(*@PROPERTIES_EX@
TYPE: POU
LOCALE: 0
IEC_LANGUAGE: ST
PLC_TYPE: independent
PROC_TYPE: independent
GROUP: AIO
*)
(*@KEY@:DESCRIPTION*)

(*@KEY@:END_DESCRIPTION*)
PROGRAM AO

(*Group:NewGroup*)

VAR
    AXL_ANALOG_OUT_1 :	AXL_ANALOG_OUT_V1_00;
END_VAR

VAR_EXTERNAL
    A07_OUT0 :	INT;
    BK_PnioDataValid :	BOOL;
    A07_IN0 :	INT;
END_VAR

VAR
    OUT1_Valid :	BOOL;
    OUT1_Status :	WORD;
    AXL_ANALOG_OUT_2 :	AXL_ANALOG_OUT_V1_00;
END_VAR

VAR_EXTERNAL
    A07_IN1 :	INT;
    A07_OUT1 :	INT;
END_VAR

VAR
    OUT2_Status :	WORD;
    OUT2_Valid :	BOOL;
    AXL_ANALOG_OUT_3 :	AXL_ANALOG_OUT_V1_00;
END_VAR

VAR_EXTERNAL
    A07_IN2 :	INT;
    A07_OUT2 :	INT;
    M :	MOTOR;
END_VAR

VAR
    OUT3_Valid :	BOOL;
    OUT3_Status :	WORD;
    AXL_ANALOG_OUT_4 :	AXL_ANALOG_OUT_V1_00;
END_VAR

VAR_EXTERNAL
    A07_OUT3 :	INT;
END_VAR

VAR
    OUT4_Valid :	BOOL;
    OUT4_Status :	WORD;
    AXL_ANALOG_OUT_5 :	AXL_ANALOG_OUT_V1_00;
END_VAR

VAR_EXTERNAL
    A07_IN4 :	INT;
END_VAR

VAR
    OUT5_Valid :	BOOL;
    OUT5_Status :	WORD;
    AXL_ANALOG_OUT_6 :	AXL_ANALOG_OUT_V1_00;
    AXL_ANALOG_OUT_7 :	AXL_ANALOG_OUT_V1_00;
    AXL_ANALOG_OUT_8 :	AXL_ANALOG_OUT_V1_00;
END_VAR

VAR_EXTERNAL
    A116_IN0 :	INT;
    A116_OUT0 :	INT;
END_VAR

VAR
    OUT6_Valid :	BOOL;
    OUT6_Status :	WORD;
END_VAR

VAR_EXTERNAL
    A116_IN1 :	INT;
    A116_OUT1 :	INT;
END_VAR

VAR
    OUT7_Valid :	BOOL;
    OUT7_Status :	WORD;
END_VAR

VAR_EXTERNAL
    A116_IN2 :	INT;
    A116_OUT2 :	INT;
END_VAR

VAR
    OUT8_Valid :	BOOL;
    OUT8_Status :	WORD;
    AXL_ANALOG_OUT_9 :	AXL_ANALOG_OUT_V1_00;
    AXL_ANALOG_OUT_10 :	AXL_ANALOG_OUT_V1_00;
END_VAR

VAR_EXTERNAL
    A116_IN3 :	INT;
END_VAR

VAR
    OUT9_Valid :	BOOL;
    OUT9_Status :	WORD;
END_VAR

VAR_EXTERNAL
    A116_IN4 :	INT;
    A116_OUT4 :	INT;
END_VAR

VAR
    OUT10_Valid :	BOOL;
    OUT10_Status :	WORD;
    AXL_ANALOG_OUT_11 :	AXL_ANALOG_OUT_V1_00;
END_VAR

VAR_EXTERNAL
    A116_IN5 :	INT;
    A116_OUT5 :	INT;
END_VAR

VAR
    OUT11_Valid :	BOOL;
    OUT11_Status :	WORD;
    AXL_ANALOG_OUT_12 :	AXL_ANALOG_OUT_V1_00;
END_VAR

VAR_EXTERNAL
    A116_IN6 :	INT;
    A116_OUT6 :	INT;
END_VAR

VAR
    OUT12_Valid :	BOOL;
    OUT12_Status :	WORD;
    AXL_ANALOG_OUT_13 :	AXL_ANALOG_OUT_V1_00;
END_VAR

VAR_EXTERNAL
    A116_IN7 :	INT;
    A116_OUT7 :	INT;
END_VAR

VAR
    OUT13_Valid :	BOOL;
    OUT13_Status :	WORD;
    AXL_ANALOG_OUT_14 :	AXL_ANALOG_OUT_V1_00;
END_VAR

VAR_EXTERNAL
    A117_IN0 :	INT;
    A117_OUT0 :	INT;
END_VAR

VAR
    OUT14_Valid :	BOOL;
    OUT14_Status :	WORD;
END_VAR

VAR_EXTERNAL
    M_AUX :	MOTOR_MISC;
END_VAR

VAR
    Blrs1_SetPower :	REAL;
    Blrs2_SetPower :	REAL;
END_VAR

VAR_EXTERNAL
    A07_IN3 :	INT;
    A07_OUT4 :	INT;
    A116_OUT3 :	INT;
END_VAR

VAR
    PmpA2_SetDose :	REAL;
    PmpA3_SetDose :	REAL;
    PmpA11_SetDose :	REAL;
    PmpA12_SetDose :	REAL;
    test :	REAL;
END_VAR

(*@KEY@: WORKSHEET
NAME: AO
IEC_LANGUAGE: ST
*)

(*============================================================================*)
    (*Boilers 1.x set power*)
(*============================================================================*)
AXL_ANALOG_OUT_1(rValue:= Blrs1_SetPower,
    rLimitLow:= 0.0,
    rLimitHigh:= 100.0,
    iRange:= 3,
    iSubstitute:= 0,
    iAnalogIn:= A07_IN0,
    xPnioDataValid:= true);

A07_OUT0:=AXL_ANALOG_OUT_1.iAnalogOut;
OUT1_Valid:=AXL_ANALOG_OUT_1.xValid;
OUT1_Status:=AXL_ANALOG_OUT_1.wStatus;

(*============================================================================*)
    (*Boilers 2.x set power*)
(*============================================================================*)
AXL_ANALOG_OUT_2(rValue:= Blrs2_SetPower,
    rLimitLow:= 0.0,
    rLimitHigh:= 100.0,
    iRange:= 3,
    iSubstitute:= 0,
    iAnalogIn:= A07_IN1,
    xPnioDataValid:= true);

A07_OUT1:=AXL_ANALOG_OUT_2.iAnalogOut;
OUT2_Valid:=AXL_ANALOG_OUT_2.xValid;
OUT2_Status:=AXL_ANALOG_OUT_2.wStatus;

(*============================================================================*)
    (*UZ5100 set frequency*)
(*============================================================================*)
AXL_ANALOG_OUT_3(rValue:= M_AUX[8].SetValue,
    rLimitLow:= 0.0,
    rLimitHigh:= 50.0,
    iRange:= 3,
    iSubstitute:= 0,
    iAnalogIn:= A07_IN2,
    xPnioDataValid:= true);

A07_OUT2:=AXL_ANALOG_OUT_3.iAnalogOut;
OUT3_Valid:=AXL_ANALOG_OUT_3.xValid;
OUT3_Status:=AXL_ANALOG_OUT_3.wStatus;

(*============================================================================*)
    (*UZ5200 set frequency*)
(*============================================================================*)
AXL_ANALOG_OUT_4(rValue:= M_AUX[9].SetValue,
    rLimitLow:= 0.0,
    rLimitHigh:= 50.0,
    iRange:= 3,
    iSubstitute:= 0,
    iAnalogIn:= A07_IN3,
    xPnioDataValid:= true);

A07_OUT3:=AXL_ANALOG_OUT_4.iAnalogOut;
OUT4_Valid:=AXL_ANALOG_OUT_4.xValid;
OUT4_Status:=AXL_ANALOG_OUT_4.wStatus;

(*============================================================================*)
    (*UZ5300 set frequency*)
(*============================================================================*)
AXL_ANALOG_OUT_5(rValue:= M_AUX[10].SetValue,
    rLimitLow:= 0.0,
    rLimitHigh:= 50.0,
    iRange:= 3,
    iSubstitute:= 0,
    iAnalogIn:= A07_IN4,
    xPnioDataValid:= true);

A07_OUT4:=AXL_ANALOG_OUT_5.iAnalogOut;
OUT5_Valid:=AXL_ANALOG_OUT_5.xValid;
OUT5_Status:=AXL_ANALOG_OUT_5.wStatus;

(*============================================================================*)
    (*UZ3100 set frequency*)
(*============================================================================*)
AXL_ANALOG_OUT_6(rValue:= M_AUX[5].SetValue,
    rLimitLow:= 0.0,
    rLimitHigh:= 50.0,
    iRange:= 3,
    iSubstitute:= 0,
    iAnalogIn:= A116_IN0,
    xPnioDataValid:= true);

A116_OUT0:=AXL_ANALOG_OUT_6.iAnalogOut;
OUT6_Valid:=AXL_ANALOG_OUT_6.xValid;
OUT6_Status:=AXL_ANALOG_OUT_6.wStatus;

(*============================================================================*)
    (*UZ3200 set frequency*)
(*============================================================================*)
AXL_ANALOG_OUT_7(rValue:= M_AUX[6].SetValue
    ,rLimitLow:= 0.0,
    rLimitHigh:= 50.0,
    iRange:= 3,
    iSubstitute:= 0,
    iAnalogIn:= A116_IN1,
    xPnioDataValid:= true);

A116_OUT1:=AXL_ANALOG_OUT_7.iAnalogOut;
OUT7_Valid:=AXL_ANALOG_OUT_7.xValid;
OUT7_Status:=AXL_ANALOG_OUT_7.wStatus;

(*============================================================================*)
    (*UZ3300 set frequency*)
(*============================================================================*)
AXL_ANALOG_OUT_8(rValue:= M_AUX[7].SetValue,
    rLimitLow:= 0.0,
    rLimitHigh:= 50.0,
    iRange:= 3,
    iSubstitute:= 0,
    iAnalogIn:= A116_IN2,
    xPnioDataValid:= true);

A116_OUT2:=AXL_ANALOG_OUT_8.iAnalogOut;
OUT8_Valid:=AXL_ANALOG_OUT_8.xValid;
OUT8_Status:=AXL_ANALOG_OUT_8.wStatus;

(*============================================================================*)
    (*UZ6100 set frequency*)
(*============================================================================*)
AXL_ANALOG_OUT_9(rValue:= M_AUX[11].SetValue,
    rLimitLow:= 0.0,
    rLimitHigh:= 50.0,
    iRange:= 3,
    iSubstitute:= 0,
    iAnalogIn:= A116_IN3,
    xPnioDataValid:= true);

A116_OUT3:=AXL_ANALOG_OUT_9.iAnalogOut;
OUT9_Valid:=AXL_ANALOG_OUT_9.xValid;
OUT9_Status:=AXL_ANALOG_OUT_9.wStatus;

(*============================================================================*)
    (*UZ6200 set frequency*)
(*============================================================================*)
AXL_ANALOG_OUT_10(rValue:= M_AUX[12].SetValue,
    rLimitLow:= 0.0,
    rLimitHigh:= 50.0,
    iRange:= 3,
    iSubstitute:= 0,
    iAnalogIn:= A116_IN4,
    xPnioDataValid:= true);

A116_OUT4:=AXL_ANALOG_OUT_10.iAnalogOut;
OUT10_Valid:=AXL_ANALOG_OUT_10.xValid;
OUT10_Status:=AXL_ANALOG_OUT_10.wStatus;

(*============================================================================*)
    (*A2 dose pump set capacity*)
(*============================================================================*)
AXL_ANALOG_OUT_11(rValue:= PmpA2_SetDose,
    rLimitLow:= 0.0,
    rLimitHigh:= 100.0,
    iRange:= 3,
    iSubstitute:= 0,
    iAnalogIn:= A116_IN5,
    xPnioDataValid:= true);

A116_OUT5:=AXL_ANALOG_OUT_11.iAnalogOut;
OUT11_Valid:=AXL_ANALOG_OUT_11.xValid;
OUT11_Status:=AXL_ANALOG_OUT_11.wStatus;

(*============================================================================*)
    (*A3 dose pump set capacity*)
(*============================================================================*)
AXL_ANALOG_OUT_12(rValue:= PmpA3_SetDose,
    rLimitLow:= 0.0,
    rLimitHigh:= 100.0,
    iRange:= 3,
    iSubstitute:= 0,
    iAnalogIn:= A116_IN6,
    xPnioDataValid:= true);

A116_OUT6:=AXL_ANALOG_OUT_12.iAnalogOut;
OUT12_Valid:=AXL_ANALOG_OUT_12.xValid;
OUT12_Status:=AXL_ANALOG_OUT_12.wStatus;

(*============================================================================*)
    (*A11 dose pump set capacity*)
(*============================================================================*)
AXL_ANALOG_OUT_13(rValue:= PmpA11_SetDose,
    rLimitLow:= 0.0,
    rLimitHigh:= 100.0,
    iRange:= 3,
    iSubstitute:= 0,
    iAnalogIn:= A116_IN7,
    xPnioDataValid:= true);

A116_OUT7:=AXL_ANALOG_OUT_13.iAnalogOut;
OUT13_Valid:=AXL_ANALOG_OUT_13.xValid;
OUT13_Status:=AXL_ANALOG_OUT_13.wStatus;

(*============================================================================*)
    (*A12 dose pump set capacity*)
(*============================================================================*)
AXL_ANALOG_OUT_14(rValue:= PmpA12_SetDose,
    rLimitLow:= 0.0,
    rLimitHigh:= 100.0,
    iRange:= 3,
    iSubstitute:= 0,
    iAnalogIn:= A117_IN0,
    xPnioDataValid:= true);

A117_OUT0:=AXL_ANALOG_OUT_14.iAnalogOut;
OUT14_Valid:=AXL_ANALOG_OUT_14.xValid;
OUT14_Status:=AXL_ANALOG_OUT_14.wStatus;

(*@KEY@: END_WORKSHEET *)
END_PROGRAM
